// TIA Portal V15 export
// export: Created 2018-12-10T18:36:42.5944446Z, ExportSetting WithDefaults, WithReadOnly, DisplayName Totally Integrated Automation Portal, DisplayVersion V15 Update 2, DisplayName TIA Portal Openness, DisplayVersion V15 Update 2, DisplayName STEP 7 Professional, DisplayVersion V15 Update 2, DisplayName STEP 7 Safety, DisplayVersion V15, DisplayName WinCC Professional, DisplayVersion V15 Update 2, DisplayName SIMATIC Visualization Architect, DisplayVersion V15 Update 1
FUNCTION "ROBNAME_Call" : Void   // FC90, FBD
TITLE = ROBNAME Station STATIONNR Robot / ROBNAME Station STATIONNR Roboter
{ S7_Optimized_Access := 'FALSE' }
VERSION : 0.1
// stored: AutoNumber true, CodeModifiedDate 2018-12-10T15:30:49.3767383Z, CompileDate 2018-12-10T15:30:49.3867136Z, CreationDate 2018-12-10T15:27:45.1479962Z, HandleErrorsWithinBlock false, InterfaceModifiedDate 2017-10-27T11:23:26.7241105Z, IsConsistent true, IsIECCheckEnabled false, IsKnowHowProtected false, IsWriteProtected false, LibraryConformanceStatus The object is library-conformant., ModifiedDate 2018-12-10T15:30:49.3767383Z, ParameterModified 2017-10-27T11:23:26.6791079Z, PLCSimAdvancedSupport false, SetENOAutomatically False, StructureModified 2017-10-27T11:23:26.7241105Z, UDAEnableTagReadback false
BEGIN
END_FUNCTION
